FUNCTION_BLOCK Sensor_Nivel_4a20_HMI (* Service Interface Function Block Type *)
  (* Standard: 61499-2 *)
  (* Version 0.0, 2/9/2026, Schneider Electric, template *)
  PACKAGE Hidryco.HidrycoLib;
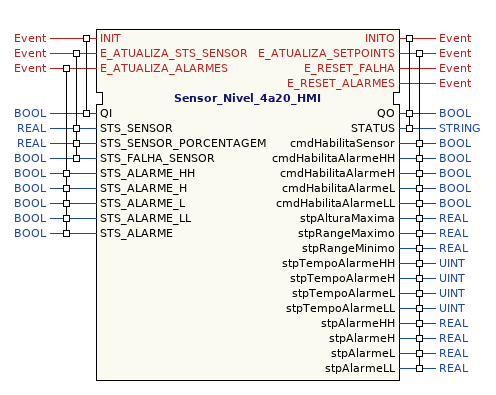
  EVENT_INPUT
    INIT WITH QI;
    E_ATUALIZA_STS_SENSOR WITH STS_SENSOR, STS_FALHA_SENSOR, STS_SENSOR_PORCENTAGEM;
    E_ATUALIZA_ALARMES WITH STS_ALARME_HH, STS_ALARME_H, STS_ALARME_L, STS_ALARME_LL, STS_ALARME;
  END_EVENT
  EVENT_OUTPUT
    INITO WITH QO, STATUS;
    E_ATUALIZA_SETPOINTS WITH cmdHabilitaSensor, cmdHabilitaAlarmeHH, cmdHabilitaAlarmeH, cmdHabilitaAlarmeL, cmdHabilitaAlarmeLL, stpAlturaMaxima, stpRangeMaximo, stpRangeMinimo, stpTempoAlarmeHH, stpTempoAlarmeH, stpTempoAlarmeL, stpTempoAlarmeLL, stpAlarmeHH, stpAlarmeH, stpAlarmeL, stpAlarmeLL;
    E_RESET_FALHA;
    E_RESET_ALARMES;
  END_EVENT
  VAR_INPUT
    QI : BOOL;
    STS_SENSOR : REAL;
    STS_SENSOR_PORCENTAGEM : REAL;
    STS_FALHA_SENSOR : BOOL;
    STS_ALARME_HH : BOOL;
    STS_ALARME_H : BOOL;
    STS_ALARME_L : BOOL;
    STS_ALARME_LL : BOOL;
    STS_ALARME : BOOL;
  END_VAR
  VAR_OUTPUT
    QO : BOOL; (* Event Output Qualifier *)
    STATUS : STRING; (* Service Status *)
    cmdHabilitaSensor : BOOL;
    cmdHabilitaAlarmeHH : BOOL;
    cmdHabilitaAlarmeH : BOOL;
    cmdHabilitaAlarmeL : BOOL;
    cmdHabilitaAlarmeLL : BOOL;
    stpAlturaMaxima : REAL;
    stpRangeMaximo : REAL;
    stpRangeMinimo : REAL;
    stpTempoAlarmeHH : UINT;
    stpTempoAlarmeH : UINT;
    stpTempoAlarmeL : UINT;
    stpTempoAlarmeLL : UINT;
    stpAlarmeHH : REAL;
    stpAlarmeH : REAL;
    stpAlarmeL : REAL;
    stpAlarmeLL : REAL;
  END_VAR
  SERVICE /
    SEQUENCE 
    END_SEQUENCE
  END_SERVICE
END_FUNCTION_BLOCK
